// TIA Portal V20 export
DATA_BLOCK "AutoIndication_DB"   // DB300
// stored: AutoNumber false, InstanceOfName AutoIndication, InstanceOfType FB
"AutoIndication"
   // VAR
   //    Var { ExternalAccessible := 'False'; ExternalVisible := 'False'; ExternalWritable := 'False'} : "TypeVar";
   //    T { ExternalAccessible := 'False'; ExternalVisible := 'False'; ExternalWritable := 'False'} : Array[1..5] of IEC_TIMER;
   // END_VAR
BEGIN
END_DATA_BLOCK
